// TIA Portal V21 program export: 0 tag tables, 0 data types, 0 data blocks, 1 code blocks (in call order from the OBs), 0 instance data blocks

ORGANIZATION_BLOCK "Main"   // OB1, LAD, ProgramCycle
TITLE = "Main Program Sweep (Cycle)"
{ S7_Optimized_Access := 'TRUE' }
VERSION : 0.1
// stored: AutoNumber true, IsIECCheckEnabled false, SetENOAutomatically false
   VAR_INPUT
      Initial_Call : Bool;
      Remanence : Bool;
   END_VAR
BEGIN

REGION Network 1: Forward interlock
   // 正转支路，反转输出作为常闭互锁。
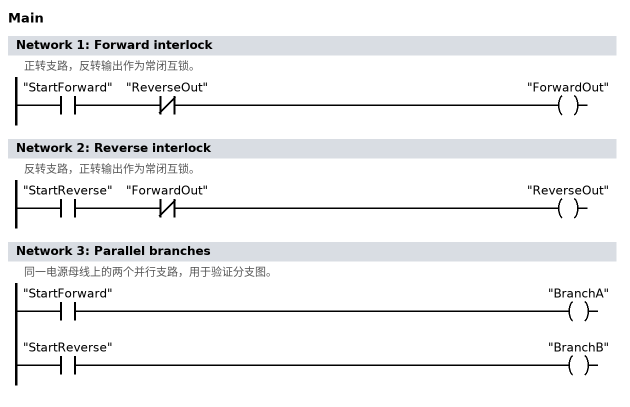
   RUNG wire#powerrail
      Contact( "StartForward" )
      I_Contact( "ReverseOut" )
      Coil( "ForwardOut" )
   END_RUNG
   // the same network as SCL:
   "ForwardOut" := "StartForward" AND NOT "ReverseOut";
END_REGION

REGION Network 2: Reverse interlock
   // 反转支路，正转输出作为常闭互锁。
   RUNG wire#powerrail
      Contact( "StartReverse" )
      I_Contact( "ForwardOut" )
      Coil( "ReverseOut" )
   END_RUNG
   // the same network as SCL:
   "ReverseOut" := "StartReverse" AND NOT "ForwardOut";
END_REGION

REGION Network 3: Parallel branches
   // 同一电源母线上的两个并行支路，用于验证分支图。
   RUNG wire#powerrail
      Contact( "StartForward" )
      Coil( "BranchA" )
   END_RUNG
   RUNG wire#powerrail
      Contact( "StartReverse" )
      Coil( "BranchB" )
   END_RUNG
   // the same network as SCL:
   "BranchA" := "StartForward";
   "BranchB" := "StartReverse";
END_REGION
END_ORGANIZATION_BLOCK
